(* LS Electric XG5000 project: 간단한프로젝트 *)
(* PLC LSPLC *)
(* module base 0 slot 0: 입력 모듈:XGI-D21A (DC 24V 입력, 8점 (전류소스/싱크입력)) *)
(* module base 0 slot 1: 출력 모듈:XGQ-RY1A (릴레이 출력, 8점 (2A용, 단독 COM.)) *)
(* module base 0 slot 2: 출력 모듈:XGQ-TR8A/B (트랜지스터 출력, 64점 (0.1A용, 싱크출력/소스출력)) *)

(* Comments on direct variables
%IX0.0.0	입력
%IX0.0.1	입력2
%IX0.0.6	실험
%QX0.1.0	출력1
%QX0.1.1	출력1-1
%QX0.1.3	출력2
%QX0.2.0	출력1-1
%QX0.2.16	출력1-2
%QX0.2.32	출력1-3
%QX0.2.48	출력1-4
*)

PROGRAM NewProgram (* task: 스캔 프로그램 *)
VAR
    출력1 : BOOL;
    출력2 : BOOL;
    출력3 : BOOL;
    출력4 : BOOL;
END_VAR

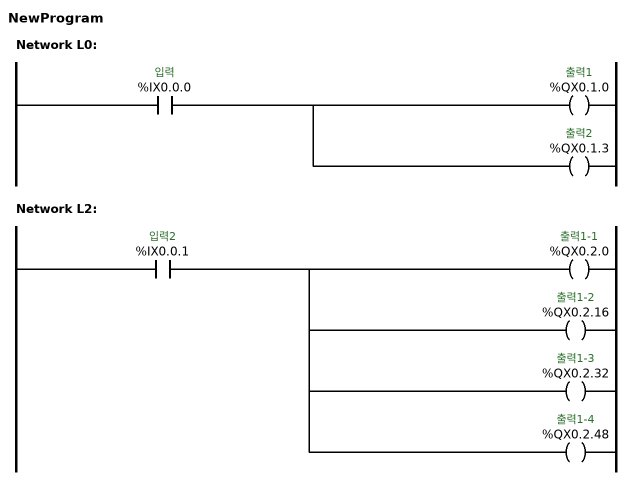
(* Rung L0 *)
%QX0.1.0 := %IX0.0.0;
%QX0.1.3 := %IX0.0.0;
(* Rung L2 *)
%QX0.2.0 := %IX0.0.1;
%QX0.2.16 := %IX0.0.1;
%QX0.2.32 := %IX0.0.1;
%QX0.2.48 := %IX0.0.1;
END_PROGRAM